TYPE ST_DigitInput :
STRUCT
	Input		: ARRAY[1..16] OF BOOL;
END_STRUCT
END_TYPE

(* stored: Version 1.1.0.1, ProductVersion 3.1.4024.9
   DUT ST_DigitInput: Id {7fd7d160-2a62-4851-8eea-174a9c184efb} *)
